FUNCTION RGBWToLED
VAR_INPUT
	RedIn	:	USINT;
	GreenIn	:	USINT;
	BlueIn	:	USINT;
	WhiteIn	:	USINT;
END_VAR
VAR_OUTPUT
	RedOut		:	INT;
	GreenOut	:	INT;
	BlueOut		:	INT;
	WhiteOut	:	INT;
END_VAR

RedOut := SingleSignalToLED(RedIn);
GreenOut := SingleSignalToLED(GreenIn);
BlueOut := SingleSignalToLED(BlueIn);
WhiteOut := SingleSignalToLED(WhiteIn);

END_FUNCTION

(* stored: Version 1.1.0.1, ProductVersion 3.1.4024.12
   POU RGBWToLED: Id {a7f06840-2832-44dc-809e-ba6984709d6c}, SpecialFunc None *)
